// TIA Portal V17 export
// export: Created 2023-04-04T07:17:24.1291369Z, ExportSetting WithDefaults, DisplayName Totally Integrated Automation Portal, DisplayVersion V17 Update 4, DisplayName TIA Portal Openness, DisplayVersion V17 Update 4, DisplayName TIA Portal Version Control Interface, DisplayVersion V17, DisplayName STEP 7 Professional, DisplayVersion V17 Update 4, DisplayName STEP 7 Safety, DisplayVersion V17, DisplayName WinCC Professional, DisplayVersion V17 Update 4
FUNCTION "PN Com Write" : Void   // FC12, LAD
TITLE = ProfiNet Data Core <-> PEMS
{ S7_Optimized_Access := 'TRUE' }
VERSION : 0.1
// stored: AutoNumber false, IsIECCheckEnabled false, SetENOAutomatically false, UDAEnableTagReadback false
BEGIN

REGION Network 1: Read & Write Data From PEMS
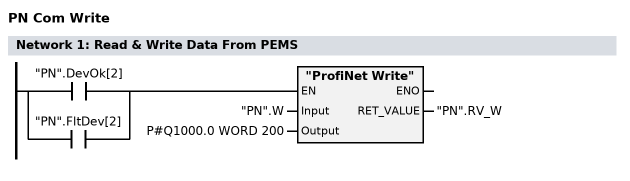
   RUNG wire#powerrail
      Contact( "PN".DevOk[2] )
      wire#w1
      "ProfiNet Write"(Input := "PN".W, Output := P#Q1000.0 WORD 200, RET_VALUE => "PN".RV_W)
   END_RUNG
   RUNG wire#powerrail
      Contact( "PN".FltDev[2] )
   END_RUNG wire#w1
   // the same network as SCL:
   IF "PN".DevOk[2] OR "PN".FltDev[2] THEN
       "ProfiNet Write"(Input := "PN".W, Output := P#Q1000.0 WORD 200, RET_VALUE => "PN".RV_W);
   END_IF;
END_REGION
END_FUNCTION
